(* CODESYS project TestSuite_V1.0.1.library
   Author: Simmel Florian
   Version: 1.0.1
   Title: Tc3PlcTestSuite
   DefaultNamespace: Tc3PlcTestSuite
   Placeholder: Tc3PlcTestSuite
   Company: Simmel

Project tree, tasks and I/O mapping:
  libraries: Tc2_Standard, * (Beckhoff Automation GmbH); Tc2_System, * (Beckhoff Automation GmbH); Tc3_EventLogger, * (Beckhoff Automation GmbH)
  Interfaces/
    interface ITestOperation: AssertEqual, ExecuteTest, State, TestId
    interface ITestSuite: Test
  Project Information/
    function F_GetCompany [ST]
    function F_GetTitle [ST]
    function F_GetVersion [ST]
  Structures/
    data type E_TestStatus
    data type ST_TestDefinition
  Version/
    global variables Global_Version
  function block FB_Test [ST]: AssertEqual, ExecuteTest, ReportAssert, State, TestId
  function block FB_TestSuite [ST]: ReRunTests, Test
  global variables TestSuite
  global variables TestSuite_Parameter
*)

// Structures/E_TestStatus
{attribute 'qualified_only'}
{attribute 'strict'}
{attribute 'to_string'}
TYPE E_TestStatus : (
		Init := 0,
		Running,
		DoneOk,
		DoneFailed
	);
END_TYPE

// Structures/ST_TestDefinition
TYPE ST_TestDefinition :
	STRUCT
		TestId : T_MaxString;
		Status : E_TestStatus;
	END_STRUCT
END_TYPE

// Version/Global_Version
{attribute 'TcGenerated'}
{attribute 'no-analysis'}
{attribute 'linkalways'}
// This function has been automatically generated from the project information.
VAR_GLOBAL CONSTANT
	{attribute 'const_non_replaced'}
	stLibVersion_Tc3PlcTestSuite : ST_LibVersion := (iMajor := 1, iMinor := 0, iBuild := 1, iRevision := 0, nFlags := 1, sVersion := '1.0.1');
END_VAR

// TestSuite
VAR_GLOBAL
	TestSuite : FB_TestSuite;
END_VAR

// TestSuite_Parameter
{attribute 'qualified_only'}
VAR_GLOBAL CONSTANT
	MaxTestCount : DINT := 10;
END_VAR

// Interfaces/ITestOperation
INTERFACE ITestOperation EXTENDS __SYSTEM.IQueryInterface

METHOD AssertEqual
VAR_INPUT
	Var1	: ANY;
	Var2	: ANY;
	Epsilon : LREAL := 0.000001;
END_VAR
END_METHOD

METHOD ExecuteTest : BOOL
VAR_INPUT
END_VAR
END_METHOD

PROPERTY State : E_TestStatus
GET
END_GET
SET
END_SET
END_PROPERTY

PROPERTY TestId : T_MaxString
GET
END_GET
SET
END_SET
END_PROPERTY

END_INTERFACE

// Interfaces/ITestSuite
INTERFACE ITestSuite EXTENDS __SYSTEM.IQueryInterface

METHOD Test : ITestOperation
VAR_INPUT
	TestId : T_MaxString;
END_VAR
END_METHOD

END_INTERFACE

// Project Information/F_GetCompany
// This function has been automatically generated from the project information.
{attribute 'signature_flag' := '1073741824'}
{attribute 'TcGenerated'}
{attribute 'no-analysis'}
FUNCTION F_GetCompany : WSTRING
VAR_INPUT
	
END_VAR

F_GetCompany := "Simmel";

END_FUNCTION

// Project Information/F_GetTitle
// This function has been automatically generated from the project information.
{attribute 'signature_flag' := '1073741824'}
{attribute 'TcGenerated'}
{attribute 'no-analysis'}
FUNCTION F_GetTitle : WSTRING
VAR_INPUT
	
END_VAR

F_GetTitle := "Tc3PlcTestSuite";

END_FUNCTION

// Project Information/F_GetVersion
// This function has been automatically generated from the project information.
{attribute 'signature_flag' := '1073741824'}
{attribute 'TcGenerated'}
{attribute 'no-analysis'}
FUNCTION F_GetVersion : ST_LibVersion
VAR_INPUT
	
END_VAR

F_GetVersion.iMajor := 1;
F_GetVersion.iMinor := 0;
F_GetVersion.iBuild := 1;
F_GetVersion.iRevision := 0;
F_GetVersion.sVersion := '1.0.1';
F_GetVersion.nFlags := 1;

END_FUNCTION

// FB_Test
FUNCTION_BLOCK FB_Test IMPLEMENTS ITestOperation
VAR
	_TestId		: T_MaxString;
	_State		: E_TestStatus;
	TestMessage : FB_TcMessage;
END_VAR

METHOD AssertEqual
VAR_INPUT
	Var1	: ANY;
	Var2	: ANY;
	Epsilon : LREAL := 0.000001;
END_VAR

VAR
	nCount	   : DINT;
	StringVar1 : T_MaxString;
	StringVar2 : T_MaxString;
	LrealVar1  : LREAL;
	LrealVar2  : LREAL;
END_VAR
IF Var1.typeclass <> Var2.typeclass THEN
	State := E_TestStatus.DoneFailed;
	ReportAssert();
	RETURN;
END_IF

IF Var1.diSize <> Var2.diSize THEN
	State := E_TestStatus.DoneFailed;
	ReportAssert();
	RETURN;
END_IF

// String
IF Var1.TypeClass = __SYSTEM.TYPE_CLASS.TYPE_ANYSTRING OR Var1.TypeClass = __SYSTEM.TYPE_CLASS.TYPE_STRING OR Var1.TypeClass = __SYSTEM.TYPE_CLASS.TYPE_WSTRING OR Var1.TypeClass = __SYSTEM.TYPE_CLASS.TYPE_XSTRING THEN
	MEMCPY(destAddr := ADR(StringVar1), srcAddr := Var1.pValue, n := DINT_TO_UDINT(Var1.diSize));
	MEMCPY(destAddr := ADR(StringVar2), srcAddr := Var2.pValue, n := DINT_TO_UDINT(Var2.diSize));
	IF StringVar1 <> StringVar2 THEN
		State := E_TestStatus.DoneFailed;
		ReportAssert();
		RETURN;
	END_IF
ELSIF Var1.TypeClass = __SYSTEM.TYPE_CLASS.TYPE_ANYREAL OR Var1.TypeClass = __SYSTEM.TYPE_CLASS.TYPE_LREAL OR Var1.TypeClass = __SYSTEM.TYPE_CLASS.TYPE_REAL THEN
	MEMCPY(destAddr := ADR(LrealVar1), srcAddr := Var1.pValue, n := DINT_TO_UDINT(Var1.diSize));
	MEMCPY(destAddr := ADR(LrealVar2), srcAddr := Var2.pValue, n := DINT_TO_UDINT(Var2.diSize));
	IF ((LrealVar1 - Epsilon) > LrealVar2) OR ((LrealVar1 + Epsilon) < LrealVar2) THEN
		State := E_TestStatus.DoneFailed;
		ReportAssert();
		RETURN;
	END_IF
ELSE
	// Byte comparison
	FOR nCount := 0 TO Var2.diSize - 1 DO
		IF Var1.pvalue[nCount] <> Var2.pvalue[nCount] THEN
			State := E_TestStatus.DoneFailed;
			ReportAssert();
			RETURN;
		END_IF
	END_FOR
END_IF

State := E_TestStatus.DoneOk;
END_METHOD

METHOD ExecuteTest : BOOL
VAR_INPUT
END_VAR
IF State = E_TestStatus.Init THEN
	State := E_TestStatus.Running;
END_IF

ExecuteTest := State = E_TestStatus.Running;
END_METHOD

METHOD PRIVATE ReportAssert
VAR
	ResultString : T_MaxString;
END_VAR
TestMessage.Create(eventClass	:= TC_EVENT_CLASSES.TestEvents,
				   nEventId		:= 1,
				   eSeverity	:= TcEventSeverity.Error,
				   ipSourceInfo := 0);

ResultString := CONCAT('Test failed - ', TestId);
TestMessage.ipArguments.AddString(ResultString);
TestMessage.Send(0);
END_METHOD

PROPERTY State :  E_TestStatus
GET
State := _State;
END_GET
SET
_State := State;
END_SET
END_PROPERTY

PROPERTY TestId : T_MaxString
GET
TestId := _TestId;
END_GET
SET
_TestId := TestId;
END_SET
END_PROPERTY

END_FUNCTION_BLOCK

// FB_TestSuite
FUNCTION_BLOCK FB_TestSuite IMPLEMENTS ITestSuite
VAR
	TestCollection	  : ARRAY[0..TestSuite_Parameter.MaxTestCount] OF FB_Test;
	NoAction		  : FB_Test := (TestId := 'No Action', State := E_TestStatus.DoneOk);
	ActiveTest		  : DINT;
	DoneMessage		  : FB_TcMessage;
	TotalTestCount	  : UDINT := 0;
	TotalOkTestCount  : UDINT := 0;
	TotalNokTestCount : UDINT := 0;
	Complete		  : BOOL;
END_VAR

METHOD ReRunTests
VAR
	i : DINT;
END_VAR
FOR i := 0 TO TestSuite_Parameter.MaxTestCount DO
	TestCollection[i].State := E_TestStatus.Init;
	ActiveTest				:= 0;
	Complete				:= FALSE;
END_FOR
END_METHOD

METHOD Test : ITestOperation
VAR_INPUT
	TestId : T_MaxString;
END_VAR

VAR
	ResultString : T_MaxString;
	i			 : DINT;
END_VAR
IF NOT Complete THEN
	FOR i := 0 TO TestSuite_Parameter.MaxTestCount DO
		// Detect first running test
		IF TestCollection[i].State = E_TestStatus.Running THEN
			ActiveTest := i;
		END_IF

		IF TestCollection[ActiveTest].State >= E_TestStatus.DoneOk THEN
			ActiveTest := 0;
		END_IF

		// Get existing Test
		IF (TestCollection[i].TestId = TestId) THEN
			IF (ActiveTest = i) OR (ActiveTest = 0) THEN
				Test := TestCollection[i];
			ELSE
				Test := NoAction;
			END_IF

			EXIT;
		END_IF

		// Add Test
		IF TestCollection[i].TestId = '' THEN
			TestCollection[i].TestId := TestId;
			Test					 := NoAction;
			EXIT;
		END_IF

		// Out of tests
		IF i = TestSuite_Parameter.MaxTestCount THEN
			Test := NoAction;
		END_IF
	END_FOR

	// Run Statistic
	TotalTestCount	  := 0;
	TotalOkTestCount  := 0;
	TotalNokTestCount := 0;
	FOR i := 0 TO TestSuite_Parameter.MaxTestCount DO
		IF TestCollection[i].TestId <> '' THEN
			TotalTestCount := TotalTestCount + 1;
			IF TestCollection[i].State = E_TestStatus.DoneOk THEN
				TotalOkTestCount := TotalOkTestCount + 1;
			END_IF

			IF TestCollection[i].State = E_TestStatus.DoneFailed THEN
				TotalNokTestCount := TotalNokTestCount + 1;
			END_IF
		END_IF
	END_FOR

	// Tests finished
	IF (TotalTestCount = (TotalOkTestCount + TotalNokTestCount)) AND NOT Complete THEN
		DoneMessage.Create(eventClass	:= TC_EVENT_CLASSES.TestEvents,
						   nEventId		:= 1,
						   eSeverity	:= TcEventSeverity.Error,
						   ipSourceInfo := 0);

		ResultString := CONCAT('Test Suite completed: ', CONCAT('Total Tests - ', TO_STRING(TotalTestCount)));
		ResultString := CONCAT(ResultString, CONCAT(', OK Tests - ', TO_STRING(TotalOkTestCount)));
		ResultString := CONCAT(ResultString, CONCAT(', Failed Tests - ', TO_STRING(TotalNokTestCount)));
		DoneMessage.ipArguments.AddString(ResultString);
		DoneMessage.Send(0);
		Complete := TRUE;
	END_IF
ELSE
	Test := NoAction;
END_IF
END_METHOD

END_FUNCTION_BLOCK
